INTERFACE IMOCK_EM


METHOD MoveDown : BOOL
VAR_INPUT
  Status : IPLCopenCall;
END_VAR
END_METHOD


METHOD MoveUp : BOOL
VAR_INPUT
  Status : IPLCopenCall;
END_VAR
END_METHOD

END_INTERFACE

(* stored: Version 1.1.0.1
   Itf IMOCK_EM: Id {ef49eb67-0dd3-08ee-1676-40a85245db25}
   Method MoveDown: Id {c1097bb8-4cd7-0965-2bad-c28e059eadf2}
   Method MoveUp: Id {b592d131-cbee-0403-212c-bb26ab20fc93} *)
